FUNCTION_BLOCK falhaFeedbackOnOff (* Composite Function Block Type *)
  (* Standard: 61499-2 *)
  (* Version 0.0, 1/26/2026, Schneider Electric, template *)
  PACKAGE Hidryco.HidrycoLib;
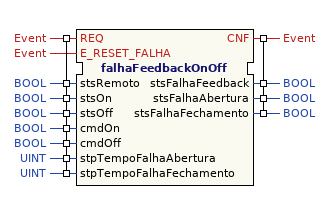
  EVENT_INPUT
    REQ WITH stsRemoto, stsOn, stsOff, cmdOn, cmdOff, stpTempoFalhaAbertura, stpTempoFalhaFechamento; (* Normal Execution Request *)
    E_RESET_FALHA;
  END_EVENT
  EVENT_OUTPUT
    CNF WITH stsFalhaFeedback, stsFalhaAbertura, stsFalhaFechamento; (* Execution Confirmation *)
  END_EVENT
  VAR_INPUT
    stsRemoto : BOOL;
    stsOn : BOOL;
    stsOff : BOOL;
    cmdOn : BOOL;
    cmdOff : BOOL;
    stpTempoFalhaAbertura : UINT;
    stpTempoFalhaFechamento : UINT;
  END_VAR
  VAR_OUTPUT
    stsFalhaFeedback : BOOL;
    stsFalhaAbertura : BOOL;
    stsFalhaFechamento : BOOL;
  END_VAR
  FBS
    FB1 : basicFalhaFeedbackOnOff;
    DelayAbertura : E_DELAYR;
    DelayFechamento : E_DELAYR;
  END_FBS
  EVENT_CONNECTIONS
    FB1.START_DELAY_ABERTURA TO DelayAbertura.RESTART;
    FB1.START_DELAY_FECHAMENTO TO DelayFechamento.RESTART;
    FB1.CNF TO CNF;
    REQ TO FB1.REQ;
    E_RESET_FALHA TO FB1.E_RESET_FALHA;
    DelayAbertura.EO TO FB1.END_DELAY_ABERTURA;
    DelayFechamento.EO TO FB1.END_DELAY_FECHAMENTO;
  END_CONNECTIONS
  DATA_CONNECTIONS
    FB1.delayTimeAbertura TO DelayAbertura.DT;
    FB1.delayTimeFechamento TO DelayFechamento.DT;
    FB1.stsFalhaFechamento TO stsFalhaFechamento;
    FB1.stsFalhaAbertura TO stsFalhaAbertura;
    FB1.stsFalhaFeedback TO stsFalhaFeedback;
    stpTempoFalhaFechamento TO FB1.stpTempoFalhaFechamento;
    stpTempoFalhaAbertura TO FB1.stpTempoFalhaAbertura;
    cmdOff TO FB1.cmdOff;
    cmdOn TO FB1.cmdOn;
    stsOff TO FB1.stsOff;
    stsOn TO FB1.stsOn;
    stsRemoto TO FB1.stsRemoto;
  END_CONNECTIONS
END_FUNCTION_BLOCK
